FUNCTION_BLOCK FBCylTronicCylinder
VAR_INPUT
	DataIn AT %I*	: CyltronicProcessDataIn;
	rSetPos			: REAL;
	rSetVelo		: REAL;
	rSetForce		: REAL;
	rSetAcc			: REAL;
	bEnable			: BOOL;
	bReset			: BOOL;
	stAxisName		: STRING;
END_VAR
VAR_OUTPUT
	DataOut AT %Q* : CyltronicProcessDataOut;
END_VAR
VAR
	bManual, bUp, bDown				: BOOL;
	UpTRIG, DownTRIG				: R_TRIG;
	iPosOffset						: INT	:= 0;
	ActualForce						: REAL;
	ActualPosition					: REAL;
	ActualSpeed						: REAL;
	LimitSwitchIn					: BOOL;
	LimitSwitchOut					: BOOL;
	MotionCommandCompleted			: BOOL;
	MotionModeActive				: BOOL;
	Ready							: BOOL;
	WarningActive					: BOOL;
	TrackingErrorToleranceExceeded	: BOOL;
	CylState						: REAL;
	Position_Aktiv					: BOOL;
	Sinus_Aktiv						: BOOL;
	BNP_Aktiv						: BOOL;
END_VAR

UpTRIG(CLK:=bUp);
DownTRIG(CLK:=bDown);

IF NOT bEnable THEN
	DataOut.CyltronicDataOutAct.MotionMode 			:= CyltronicMotionMode.Off;
	DataOut.CyltronicDataOutAct.TargetPosition 		:= DataIn.CyltronicDataInAct.ActualPosition;
	bManual 										:= FALSE;
ELSIF bReset THEN
	DataOut.CyltronicDataOutAct.MotionMode			:= CyltronicMotionMode.Reset;
	bReset 											:= FALSE;
ELSIF NOT bManual THEN
	DataOut.CyltronicDataOutAct.TargetPosition		:= LIMIT(0,rSetPos,MaxTravel);
	DataOut.CyltronicDataOutAct.MotionMode			:= CyltronicMotionMode.FreePosPro;
ELSE
	IF UpTrig.Q AND iPosOffset < MaxTravel THEN
		iPosOffset := iPosOffset + GVL.StepSize;
	ELSIF DownTrig.Q AND iPosOffset > - MaxTravel THEN
		iPosOffset := iPosOffset - GVL.StepSize;
	END_IF
	DataOut.CyltronicDataOutAct.TargetPosition		:= LIMIT(0,rSetPos + iPosOffset,MaxTravel);
	DataOut.CyltronicDataOutAct.MotionMode			:= CyltronicMotionMode.FreePosPro;
	iPosOffset := 0;
END_IF

//Outputs
DataOut.CyltronicDataOutAct.AccelerationOverride 	:= LIMIT(1, REAL_TO_USINT(rSetAcc / MaxACC * 100), 255);
DataOut.CyltronicDataOutAct.ForceOverride 			:= LIMIT(1, REAL_TO_USINT(rSetForce / MaxForce * 100), 255);
DataOut.CyltronicDataOutAct.SpeedOverride 			:= LIMIT(1, REAL_TO_USINT(rSetVelo / MaxVelo * 100), 255);

ActualForce											:= DataIn.CyltronicDataInAct.ActualForce;
ActualPosition										:= DataIn.CyltronicDataInAct.ActualPosition;
ActualSpeed											:= DataIn.CyltronicDataInAct.ActualSpeed;
LimitSwitchIn										:= DataIn.CyltronicDataInAct.LimitSwitchIn;
LimitSwitchOut										:= DataIn.CyltronicDataInAct.LimitSwitchOut;
MotionCommandCompleted								:= DataIn.CyltronicDataInAct.MotionCommandCompleted;
MotionModeActive									:= DataIn.CyltronicDataInAct.MotionModeActive;
Ready												:= DataIn.CyltronicDataInAct.Ready;
WarningActive										:= DataIn.CyltronicDataInAct.WarningActive;
TrackingErrorToleranceExceeded						:= DataIn.CyltronicDataInAct.TrackingErrorToleranceExceeded;
CylState											:= DataIn.CyltronicDataInAct.State;

END_FUNCTION_BLOCK

(* stored: Version 1.1.0.1, ProductVersion 3.1.4024.10
   POU FBCylTronicCylinder: Id {065cd091-3563-4a4f-b586-4eea2d97404e}, SpecialFunc None *)
